// TIA Portal project "第二节课学习置位复位2" (V15.1)

(* hardware
DEVICE "S7-1200 station_1"  S7-1200 Station
   slot 0: "Rack_0"  S7-1200 Rack  Rack  V1.0
   slot 1: "PLC_1"  CPU 1212C DC/DC/DC  6ES7 212-1AE40-0XB0  V4.2
*)

// ===== PLC "PLC_1"  CPU 1212C DC/DC/DC =====

VAR_GLOBAL   // PLC tag table "io"
   "启动" AT %I0.0 : Bool;
   "中间标志" AT %M0.0 : Bool;
   "关闭" AT %I0.1 : Bool;
   "启动1" AT %I0.2 : Bool;
   "关闭1" AT %I0.3 : Bool;
   "中间标志(1)" AT %M0.1 : Bool;
END_VAR

ORGANIZATION_BLOCK "Main"   // OB1, LAD, ProgramCycle
TITLE = "Main Program Sweep (Cycle)"
{ S7_Optimized_Access := 'TRUE' }
VERSION : 0.1
   VAR_INPUT
      Initial_Call : Bool;   // Initial call of this OB
      Remanence : Bool;   // =True, if remanent data are available
   END_VAR
BEGIN

REGION Network 1
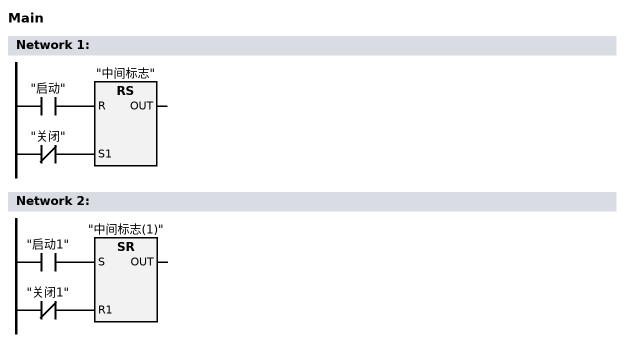
   RUNG wire#powerrail
      Contact( "启动" )
      S_RS(operand := "中间标志", s1 := wire#w1)
   END_RUNG
   RUNG wire#powerrail
      I_Contact( "关闭" )
   END_RUNG wire#w1
   // the same network as SCL:
   IF "启动" THEN
       "中间标志" := FALSE;   // RS flip-flop
   END_IF;
   IF NOT "关闭" THEN "中间标志" := TRUE; END_IF;
END_REGION

REGION Network 2
   RUNG wire#powerrail
      Contact( "启动1" )
      S_SR(operand := "中间标志(1)", r1 := wire#w1)
   END_RUNG
   RUNG wire#powerrail
      I_Contact( "关闭1" )
   END_RUNG wire#w1
   // the same network as SCL:
   IF "启动1" THEN
       "中间标志(1)" := TRUE;   // SR flip-flop
   END_IF;
   IF NOT "关闭1" THEN "中间标志(1)" := FALSE; END_IF;
END_REGION
END_ORGANIZATION_BLOCK